(* PLC project Test, D OpenPLC 1.0 *)
(* stored: creationDateTime 2018-09-26T00:48:44, modificationDateTime 2018-10-04T02:42:53 *)

PROGRAM Test_Program
  VAR
    ESP0 AT %QX0.0 : BOOL;
    TMP AT %QX0.2 : BOOL;
    ESP1 AT %QX0.1 : BOOL;
  END_VAR
  VAR
    TON1 : TON;
    TON2 : TON;
  END_VAR

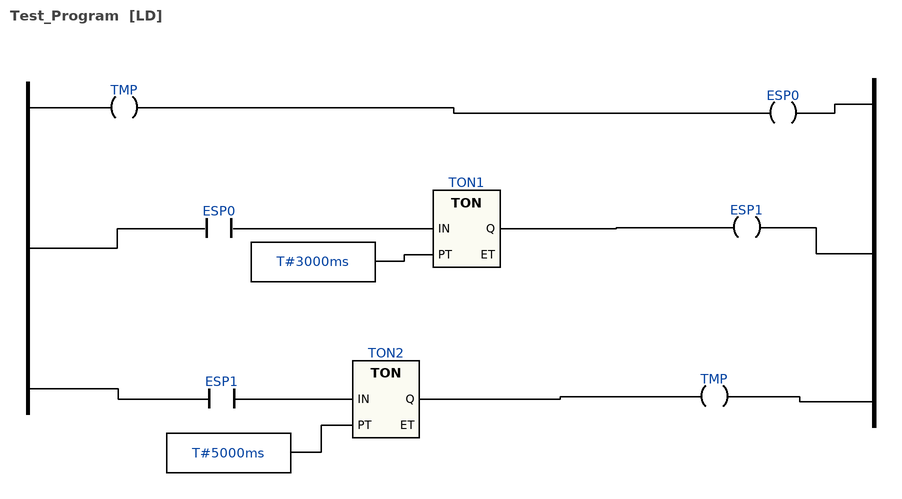
(* LD diagram, written out as Structured Text *)
TMP := TRUE;
ESP0 := TRUE;
TON1(IN := ESP0, PT := T#3000ms);
ESP1 := TON1.Q;
TON2(IN := ESP1, PT := T#5000ms);
TMP := TON2.Q;
END_PROGRAM

CONFIGURATION Config0
  RESOURCE Res0 ON PLC
    TASK MyTask(INTERVAL := T#50ms, PRIORITY := 0);
    PROGRAM instance0 WITH MyTask : Test_Program;
  END_RESOURCE
END_CONFIGURATION
